FUNCTION_BLOCK FB_ActionTestObject EXTENDS TcBase.FB_OrphanObject IMPLEMENTS TcBase.I_CyclicTask
VAR
    _nCounter: UDINT;
    _bActivated: BOOL;
END_VAR

METHOD Activate
VAR_INPUT
    bActivate: BOOL;
END_VAR
THIS^._bActivated := bActivate;
END_METHOD

PROPERTY bIsActivated : BOOL
GET
bIsActivated := THIS^._bActivated;
END_GET
END_PROPERTY

PROPERTY nCounter : UDINT
GET
nCounter := THIS^._nCounter;
END_GET
END_PROPERTY

METHOD Run
VAR_INPUT
END_VAR
THIS^._nCounter := THIS^._nCounter + 1;
END_METHOD

END_FUNCTION_BLOCK

(* stored: Version 1.1.0.1, ProductVersion 3.1.4024.12
   POU FB_ActionTestObject: Id {037c4d37-edf6-44b1-862b-4f277bf61049}, SpecialFunc None
   Method Activate: Id {7eb5a50d-f174-4a26-bdbd-2b872425447b}
   Property bIsActivated: Id {6b4c44f8-0292-48e4-9999-9b92593cc480}
   Get Get: Id {a11589de-a08c-4a47-a2f4-0dfa8196207c}
   Property nCounter: Id {25e1eae1-e6f7-422c-846f-9d23f9f31c73}
   Get Get: Id {92b34af0-f419-439d-a4f3-6ac36d83b60f}
   Method Run: Id {80772e95-86c4-4e9d-b664-656b36756d5e} *)
